// TIA Portal V19 export
TYPE "PNOZ Comm"
TITLE = Connection Parameters for TCON
   STRUCT
      block_length : Word := WORD#16#0040;   // #!PNOZ m ES ETH!#
      id : Word := WORD#16#0002;
      connection_type : Byte := BYTE#16#11;
      active_est : Bool := TRUE;
      local_device_id : Byte := BYTE#16#03;
      local_tsap_id_len : Byte;
      rem_subnet_id_len : Byte;
      rem_staddr_len : Byte := BYTE#16#04;
      rem_tsap_id_len : Byte := BYTE#16#02;
      next_staddr_len : Byte;
      local_tsap_id : Array[1..16] of Byte;
      rem_subnet_id : Array[1..6] of Byte;
      rem_staddr : Array[1..6] of Byte;
      rem_tsap_id : Array[1..16] of Byte;
      next_staddr : Array[1..6] of Byte;
      spare : Word;   // #!PNOZ m ES ETH!#
   END_STRUCT;
   // rem_staddr[1] := BYTE#16#A9;
   // rem_staddr[2] := BYTE#16#FE;
   // rem_staddr[3] := BYTE#16#3C;
   // rem_staddr[4] := BYTE#16#01;
   // rem_tsap_id[1] := BYTE#16#23;
   // rem_tsap_id[2] := BYTE#16#28;
END_TYPE
